PROGRAM MAIN
VAR
END_VAR

END_PROGRAM

(* stored: Version 1.1.0.1
   POU MAIN: Id {13717ce7-e361-49d8-94c5-d36f6433cb71} *)
